FUNCTION_BLOCK FB_RecordValue
VAR_INPUT
END_VAR
VAR_OUTPUT
END_VAR
VAR
END_VAR

END_FUNCTION_BLOCK

(* stored: Version 1.1.0.1, ProductVersion 3.1.4026.18
   POU FB_RecordValue: Id {43532e2a-7bcc-4fae-9ce2-8f1c24dbad4d}, SpecialFunc None *)
